// TIA Portal V20 export
DATA_BLOCK "System_To_Moving_Pallets_DB"   // DB25
// stored: InstanceOfName System_To_Moving_Pallets, InstanceOfType FB
"System_To_Moving_Pallets"
   // VAR
   //    iCenterTippler : Bool;
   //    oCeterTippler : Bool;
   //    Reset_Centering_Tippler : Bool;
   //    ST13_ST14 { S7_SetPoint := 'True'} : "Pallet_Transport_Row_4";
   //    ST12_ST13 { S7_SetPoint := 'True'} : "Pallet_Transport_Row_4";
   //    ST11_ST12 { S7_SetPoint := 'True'} : "Pallet_Transport_Row_4";
   //    ST10_ST11 { S7_SetPoint := 'True'} : "Pallet_Transport_Row_4";
   //    ST09_ST10 { S7_SetPoint := 'True'} : "Pallet_Transport_Row_4";
   //    ST08_ST09 { S7_SetPoint := 'True'} : "Pallet_Transport_Row_4";
   //    ST07_ST08 { S7_SetPoint := 'True'} : "Pallet_Transport_Row_4";
   //    ST06_ST07 { S7_SetPoint := 'True'} : "Pallet_Transport_Row_4";
   //    ST05_ST06 { S7_SetPoint := 'True'} : "Pallet_Transport_Row_4";
   //    ST04_ST05 { S7_SetPoint := 'True'} : "Pallet_Transport_Row_4";
   //    ST01_ST02 { S7_SetPoint := 'True'} : "Pallet_Transport_Row_1_2";
   //    ST02_ST01 { S7_SetPoint := 'True'} : "Pallet_Transport_Row_1_2";
   //    ST38_ST01 { S7_SetPoint := 'True'} : "Pallet_Transport_Row_1_2";
   //    ST01_ST38 { S7_SetPoint := 'True'} : "Pallet_Transport_Row_1_2";
   //    ST34_ST35 { S7_SetPoint := 'True'} : "Pallet_Transport_Row_1_2";
   //    ST35_ST34 { S7_SetPoint := 'True'} : "Pallet_Transport_Row_1_2";
   //    ST33_ST34 { S7_SetPoint := 'True'} : "Pallet_Transport_Row_1_2";
   //    ST34_ST33 { S7_SetPoint := 'True'} : "Pallet_Transport_Row_1_2";
   //    ST32_ST33 { S7_SetPoint := 'True'} : "Pallet_Transport_Row_1_2";
   //    ST36_ST38 { S7_SetPoint := 'True'} : "Pallet_Transport_Row_1_2";
   //    ST38_ST36 { S7_SetPoint := 'True'} : "Pallet_Transport_Row_1_2";
   //    ST37_ST36 { S7_SetPoint := 'True'} : "Pallet_Transport_Row_1_2";
   //    ST18_ST37 { S7_SetPoint := 'True'} : "Pallet_Transport_Row_1_2";
   //    ST19_ST18 { S7_SetPoint := 'True'} : "Pallet_Transport_Row_1_2";
   //    ST20_ST19 { S7_SetPoint := 'True'} : "Pallet_Transport_Row_1_2";
   //    ST21_ST20 { S7_SetPoint := 'True'} : "Pallet_Transport_Row_1_2";
   //    ST22_ST21 { S7_SetPoint := 'True'} : "Pallet_Transport_Row_1_2";
   //    ST23_ST22 { S7_SetPoint := 'True'} : "Pallet_Transport_Row_1_2";
   //    ST24_ST23 { S7_SetPoint := 'True'} : "Pallet_Transport_Row_1_2";
   //    Centering_Perform : Array[7..13, 1..3] of Bool;
   //    Centering_Status { S7_SetPoint := 'True'} : Array[7..13, 1..3] of Bool;
   //    ST31_ST32 { S7_SetPoint := 'True'} : "Pallet_Transport_Row_1_2";
   //    ST30_ST31 { S7_SetPoint := 'True'} : "Pallet_Transport_Row_1_2";
   //    ST29_ST30 { S7_SetPoint := 'True'} : "Pallet_Transport_Row_1_2";
   //    ST28_ST29 { S7_SetPoint := 'True'} : "Pallet_Transport_Row_1_2";
   //    TON_Reset_Drives { S7_SetPoint := 'True'} : TON_TIME;
   //    TP_Reset_Drives { S7_SetPoint := 'True'} : TP_TIME;
   //    Reset_Drives_Var { S7_SetPoint := 'True'} : Bool;
   //    ST27_ST28 { S7_SetPoint := 'True'} : "Pallet_Transport_Row_1_2";
   //    ST26_ST27 { S7_SetPoint := 'True'} : "Pallet_Transport_Row_1_2";
   //    ST25_ST26 { S7_SetPoint := 'True'} : "Pallet_Transport_Row_1_2";
   //    tComm_W1 { S7_SetPoint := 'True'} : TON_TIME;
   //    tComm_W2 { S7_SetPoint := 'True'} : TON_TIME;
   //    tComm_W4 { S7_SetPoint := 'True'} : TON_TIME;
   // END_VAR
BEGIN
END_DATA_BLOCK
